Universal Robots PolyScope program: dummy step right.urp

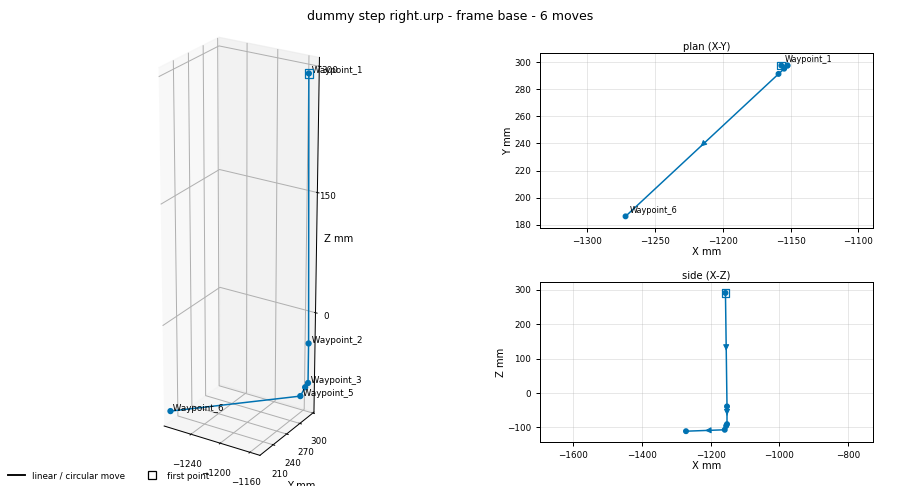
[picture p0: tool path of dummy step right.urp in frame base, 6 of 6 moves have a stored position in this frame; points joined in program order, loops and branches not executed]
Program dummy step right (installation=default directory=/programs createdIn=5.21.3 lastSavedIn=5.21.3 robotSerialNumber=20246801938)
Calibrated DH parameters: a=[-0.000071, -0.790281, -0.600694, 0.000061, -0.000039, 0]; d=[0.236272, 604.465945, 132.116513, -736.382239, 0.159268, 0.154005]; alpha=[1.570254, -0.000567, 0.000559, 1.571709, -1.56999, 0]; deltaTheta=[0, -0.409357, 7.293326, -0.600784, -0.000001, -0.000001]
InitVariablesNode
Robot Program (runOnlyOnce=true)
  MoveJ speed 60 deg/s, acceleration 80 deg/s^2 (useActiveTCP=true optimoveEnabled=false optiMoveSpeed=0.3 optiMoveAcceleration=0.09) feature=Base
    Waypoint Waypoint_1: TCP in base x=-1156.816 y=297.468 z=291.375 mm, rx=-0.7812 ry=-1.774 rz=1.7129 rad; joints [-189.786, -111.954, -118.346, -130.254, -52.7, 88.101] deg; TCP offset x=-9.5 y=-328 z=105.73 mm, rx=1.2092 ry=-1.2092 rz=1.2092 rad
  MoveP speed 10 mm/s, acceleration 1200 mm/s^2 (blendRadius=0.025 useActiveTCP=true optimoveEnabled=false optiMoveSpeed=0.3 optiMoveAcceleration=0.09) feature=Base
    Waypoint Waypoint_2: TCP in base x=-1152.293 y=297.468 z=-38.814 mm, rx=-0.7812 ry=-1.774 rz=1.7129 rad; joints [-189.832, -134.502, -121.263, -104.779, -52.744, 88.083] deg
    Waypoint Waypoint_3: TCP in base x=-1152.293 y=297.468 z=-90.397 mm, rx=-0.7812 ry=-1.774 rz=1.7129 rad; joints [-189.83, -138.406, -120.62, -101.517, -52.743, 88.081] deg
  MoveP speed 2 mm/s, acceleration 100 mm/s^2 (blendRadius=0.001 useActiveTCP=true optimoveEnabled=false optiMoveSpeed=0.3 optiMoveAcceleration=0.09) feature=Base
    Waypoint Waypoint_4: motionParameters(blendRadius=0); TCP in base x=-1154.733 y=295.137 z=-95.599 mm, rx=-0.4323 ry=-0.9675 rz=2.1538 rad; joints [-185.377, -156.212, -111.627, -92.731, -48.297, 131.757] deg
    Waypoint Waypoint_5: TCP in base x=-1158.881 y=291.274 z=-106.746 mm, rx=-0.0236 ry=-0.0268 rz=2.3202 rad; joints [-174.705, -165.939, -94.699, -100.058, -37.633, 178.995] deg
  MoveL speed 10 mm/s, acceleration 1200 mm/s^2 (useActiveTCP=true optimoveEnabled=false optiMoveSpeed=0.3 optiMoveAcceleration=0.09) feature=Base
    Waypoint Waypoint_6: TCP in base x=-1271.643 y=186.285 z=-110.88 mm, rx=-0.0236 ry=-0.0268 rz=2.3202 rad; joints [-169.654, -167.895, -84.476, -108.42, -32.586, 179.114] deg
